// TIA Portal V18 export
DATA_BLOCK "monitor_perifery_DB"   // DB15
VERSION : 0.1
// stored: AutoNumber true, DBAccessibleFromOPCUA true, InstanceOfName monitor_perifery, InstanceOfType FB
"monitor_perifery"
   // VAR_INPUT
   //    ptDelayed : Time;
   //    inWord : Byte;
   //    ptMax : Time;
   //    xBitON : Bool;
   // END_VAR
   // VAR_OUTPUT
   //    outWord : Byte;
   //    yERCOMM : Bool;
   //    yWNdelay : Bool;
   //    yAllModulesLive : Bool;
   // END_VAR
   // VAR
   //    IEC_Timer_0_Instance { S7_SetPoint := 'True'} : TON_TIME;
   //    startup { S7_SetPoint := 'True'} : TON_TIME;
   //    delayPassed : Bool;
   // END_VAR
BEGIN
END_DATA_BLOCK
